(* PLC project Plc1, Beckhoff Automation GmbH TwinCAT PLC Control 3.5.13.21 *)
(* stored: creationDateTime 2025-06-23T09:46:51.3138385, modificationDateTime 2025-06-23T09:46:51.3178282 *)

TYPE ST_CompleteSystemState :
STRUCT
	Motor : ST_Motor;
	Lights : ST_LightSystem;
END_STRUCT
END_TYPE

TYPE ST_Light :
STRUCT
	STATE : BOOL;
	COLOR : STRING(10);
	LAST_TRIGGERED : STRING(30);
END_STRUCT
END_TYPE

TYPE ST_LightSystem :
STRUCT
	LIGHT1 : ST_Light;
	LIGHT2 : ST_Light;
	LIGHT3 : ST_Light;
END_STRUCT
END_TYPE

TYPE ST_LightSystemWithHistory :
STRUCT
	LightSystem : ST_LightSystem;
END_STRUCT
END_TYPE

TYPE ST_Motor :
STRUCT
	STATE : BOOL;
	SPEED : REAL := GVL.defaultSpeed;
END_STRUCT
END_TYPE

FUNCTION CheckIfUpdatedLight : BOOL
VAR_INPUT
	RealTimeState : ST_LightSystem;
	ReadState : ST_LightSystem;
END_VAR
VAR
END_VAR

                  IF (RealTimeState.LIGHT1.STATE <> ReadState.LIGHT1.STATE) OR
	(RealTimeState.LIGHT2.STATE <> ReadState.LIGHT2.STATE) OR
	(RealTimeState.LIGHT3.STATE <> ReadState.LIGHT3.STATE) THEN
	CheckIfUpdatedLight := TRUE;
ELSE
	CheckIfUpdatedLight := FALSE;
END_IF
                
END_FUNCTION

FUNCTION GetTimeAsString : STRING
VAR_INPUT
END_VAR
VAR
	fbSystemTime : GETSYSTEMTIME;
    timeAsFileTime : T_FILETIME;
END_VAR

                  fbSystemTime(
    timeLoDW=>timeAsFileTime.dwLowDateTime,
    timeHiDW=>timeAsFileTime.dwHighDateTime );
GetTimeAsString := DT_TO_STRING(FILETIME_TO_DT(timeAsFileTime));
                
END_FUNCTION

FUNCTION_BLOCK MotorProps
VAR_INPUT
	Motor : REFERENCE TO ST_Motor;
	MotorSpeed : REAL := 500;
END_VAR
VAR_OUTPUT
END_VAR
VAR
END_VAR

                  IF Motor.STATE THEN
	Motor.SPEED := MotorSpeed;
ELSE
	Motor.SPEED := 0;
END_IF
                
END_FUNCTION_BLOCK

FUNCTION CheckIfUpdatedMotor : BOOL
VAR_INPUT
	RealTimeState : ST_Motor;
	ReadState : ST_Motor;
END_VAR
VAR
END_VAR

                  IF (RealTimeState.SPEED <> ReadState.SPEED) OR
	(RealTimeState.STATE <> ReadState.STATE) THEN
	CheckIfUpdatedMotor := TRUE;
ELSE
	CheckIfUpdatedMotor := FALSE;
END_IF
                
END_FUNCTION

PROGRAM MAIN
VAR
	// relating to light system
	GreenLight : ST_Light := (COLOR := 'GREEN');
	BlueLight : ST_Light := (COLOR := 'BLUE');
	YellowLight : ST_Light := (COLOR := 'YELLOW');
	GBY_LightSystem : ST_LightSystem := (LIGHT1:= GreenLight, 
										LIGHT2 := BlueLight,
										LIGHT3 := YellowLight);
	GreenToggle : BOOL;
	BlueToggle : BOOL;
	YellowToggle : BOOL;
	bExecuteLight : BOOL;
										
	// relating to motor system
	stMotor : ST_Motor;
	MotorToggle : BOOL := FALSE;
	bExecuteMotor : BOOL := FALSE;
	fbMotor : MotorProps;
	
	// writing xml files
//	CurrentStateFileNameMotor : T_MaxString := 'CurrentLightSystem.xml';
//	RealTimeStateOfMotor : ST_MotorSystem;
//	XmlSrvWriteSystemCurrentStateOfMotor : FB_XmlSrvWrite := (nMode := XMLSRV_ADDMISSING,
//														pSymAddr:=ADR(RealTimeStateOfMotor),
//														cbSymSize := SIZEOF(RealTimeStateOfMotor),
//														sFilePath := CONCAT(STR1:=GVL.BasePath, STR2:=CurrentStateFileNameMotor),
//														sXPath := '/CURRENT_STATE/Motor');
														
//	CurrentStateFileNameLight : T_MaxString := 'CurrentLightSystem.xml';
//	RealTimeStateOfLight : ST_LightSystem;
//	XmlSrvWriteSystemCurrentStateOfLight : FB_XmlSrvWrite := (nMode := XMLSRV_ADDMISSING,
//														pSymAddr:=ADR(RealTimeStateOfLight),
//														cbSymSize := SIZEOF(RealTimeStateOfLight),
//														sFilePath := CONCAT(STR1:=GVL.BasePath, STR2:=CurrentStateFileNameLight),
//														sXPath := '/CURRENT_STATE/Lights');
	CurrentStateFileNameMotor : T_MaxString := 'CurrentSystem.xml';
	RealTimeStateOfSystem : ST_CompleteSystemState;
	XmlSrvWriteSystemCurrentStateOfSystem : FB_XmlSrvWrite := (nMode := XMLSRV_ADDMISSING,
														pSymAddr:=ADR(RealTimeStateOfSystem),
														cbSymSize := SIZEOF(RealTimeStateOfSystem),
														sFilePath := CONCAT(STR1:=GVL.BasePath, STR2:=CurrentStateFileNameMotor),
														sXPath := '/CURRENT_STATE');

	// write logs
	CurrentStateFileNameLightHistory : T_MaxString := 'LightHistory.xml';
	RealTimeLightSystemHistory : ST_LightSystemWithHistory;
//	RealTimeLightSystemHistory : ST_LightSystemWithHistory := (LightSystem.LIGHT1 := GreenLight,
//																LightSystem.LIGHT2 := BlueLight,
//																LightSystem.LIGHT3 := YellowLight);		
	XmlSrvWriteSystemCurrentStateOfLightAndHistory : FB_XmlSrvWrite := (nMode := XMLSRV_ADDMISSING,
														pSymAddr:=ADR(RealTimeLightSystemHistory),
														cbSymSize := SIZEOF(RealTimeStateOfSystem.Lights),
														sFilePath := CONCAT(STR1:=GVL.BasePath, STR2:=CurrentStateFileNameLightHistory));										
	iStateIndex : UDINT := 0;
	
	// read xml files
	// read xml file from 'CurrentSystemState.xml'
	ReadStateOfSystem : ST_CompleteSystemState;
	XmlSrvReadCurrentSystemStateOfSystem : FB_XmlSrvRead := (pSymAddr := ADR(ReadStateOfSystem),
											cbSymSize := SIZEOF(ReadStateOfSystem),
											sFilePath := CONCAT(STR1:=GVL.BasePath, STR2:=CurrentStateFileNameMotor),
											sXPath := '/CURRENT_STATE');
											
//	ReadStateOfMotor : ST_Motor;
//	XmlSrvReadCurrentSystemStateMotor : FB_XmlSrvRead := (pSymAddr := ADR(ReadStateOfMotor),
//											cbSymSize := SIZEOF(ReadStateOfMotor),
//											sFilePath := CONCAT(STR1:=GVL.BasePath, STR2:=CurrentStateFileNameMotor),
//											sXPath := '/CURRENT_STATE/Motor');
											
											
    Timer3Sec : TON;
    Pulse : BOOL := FALSE;
	
	oldState: BOOL := FALSE;
	MotorStateChanged : BOOL := FALSE;
	
	tempVar : BOOL;
END_VAR

                  Timer3Sec(IN := TRUE, PT := T#1500MS);
IF Timer3Sec.Q THEN
    Pulse := TRUE;
    Timer3Sec(IN := FALSE);
ELSE
    Pulse := FALSE;
END_IF;

IF GreenToggle THEN
	GreenLight.STATE := NOT GreenLight.STATE;
	GBY_LightSystem.LIGHT1:=GreenLight;
	RealTimeLightSystemHistory.LightSystem.LIGHT1.LAST_TRIGGERED := GetTimeAsString();
	bExecuteLight := TRUE;
END_IF
IF BlueToggle THEN
	BlueLight.STATE := NOT BlueLight.STATE;
	GBY_LightSystem.LIGHT2:=BlueLight;
	RealTimeLightSystemHistory.LightSystem.LIGHT2.LAST_TRIGGERED := GetTimeAsString();
	bExecuteLight := TRUE;
END_IF
IF YellowToggle THEN
	YellowLight.STATE := NOT YellowLight.STATE;
	GBY_LightSystem.LIGHT3:=YellowLight;
	RealTimeLightSystemHistory.LightSystem.LIGHT3.LAST_TRIGGERED := GetTimeAsString();
	bExecuteLight := TRUE;
END_IF

fbMotor(Motor := stMotor, MotorSpeed := ReadStateOfSystem.Motor.SPEED);
IF oldState <> MotorToggle THEN
	MotorStateChanged := TRUE;
END_IF
IF MotorStateChanged THEN
	stMotor.STATE := NOT stMotor.STATE;
	bExecuteMotor := TRUE;
END_IF
oldState := MotorToggle;

// update system state variable
RealTimeStateOfSystem.Lights := GBY_LightSystem;
RealTimeStateOfSystem.Motor := stMotor;

// write xml files
IF (bExecuteLight OR bExecuteMotor) AND NOT XmlSrvWriteSystemCurrentStateOfSystem.bBusy THEN
	XmlSrvWriteSystemCurrentStateOfSystem(pSymAddr := ADR(RealTimeStateOfSystem), bExecute := TRUE);
ELSE
	XmlSrvWriteSystemCurrentStateOfSystem(pSymAddr := ADR(RealTimeStateOfSystem), bExecute := FALSE);
END_IF

IF (bExecuteLight) AND NOT XmlSrvWriteSystemCurrentStateOfLightAndHistory.bBusy THEN
	XmlSrvWriteSystemCurrentStateOfLightAndHistory(sXPath := CONCAT('/STATE_LOG/STATE_', 
																	UDINT_TO_STRING(iStateIndex) ),
												pSymAddr := ADR(RealTimeLightSystemHistory), 
												bExecute := TRUE);
	iStateIndex := iStateIndex + 1;
ELSE
	XmlSrvWriteSystemCurrentStateOfLightAndHistory(sXPath := CONCAT('/STATE_LOG/STATE_', 
																	UDINT_TO_STRING(iStateIndex) ),
												pSymAddr := ADR(RealTimeLightSystemHistory), 
												bExecute := FALSE);
END_IF

// read xml files
IF NOT XmlSrvReadCurrentSystemStateOfSystem.bBusy AND NOT XmlSrvWriteSystemCurrentStateOfSystem.bBusy AND Pulse THEN
	XmlSrvReadCurrentSystemStateOfSystem(bExecute := TRUE);
ELSIF XmlSrvReadCurrentSystemStateOfSystem.bBusy THEN
	XmlSrvReadCurrentSystemStateOfSystem(bExecute := FALSE);
END_IF

// check if xml files are updated
IF CheckIfUpdatedLight(RealTimeStateOfSystem.Lights, ReadStateOfSystem.Lights) AND Pulse THEN
	GBY_LightSystem := ReadStateOfSystem.Lights;
END_IF
IF CheckIfUpdatedMotor(RealTimeStateOfSystem.Motor, ReadStateOfSystem.Motor) AND Pulse THEN
	stMotor.SPEED := ReadStateOfSystem.Motor.SPEED;
	stMotor.STATE := ReadStateOfSystem.Motor.STATE;
	IF ReadStateOfSystem.Motor.STATE = FALSE THEN
		stMotor.SPEED := 0;
	END_IF
END_IF

GreenToggle := FALSE;
BlueToggle := FALSE;
YellowToggle := FALSE;
bExecuteLight := FALSE;
bExecuteMotor := FALSE;
MotorStateChanged := FALSE;
//tempVar := FALSE;
                
END_PROGRAM

CONFIGURATION Application
  RESOURCE Plc1 ON PLC
(* global variable list GVL *)
{attribute 'qualified_only'}
VAR_GLOBAL
	BasePath : T_MaxString := 'C:\Users\suura\Desktop\';
	defaultSpeed : REAL := 500;
END_VAR
    TASK PlcTask(INTERVAL := T#0ms, PRIORITY := 20);
    PROGRAM MAIN WITH PlcTask : MAIN;
  END_RESOURCE
END_CONFIGURATION
